# EPICS autosave request: iocBoot/sioc-li21-im01/adc_manual.req
file "manual.req" AREA=IN20,POS=432
file "manual.req" AREA=IN20,POS=792
file "manual.req" AREA=IN20,POS=972
file "manual.req" AREA=IN20,POS=216
